TYPE ST_CX_EtherCATMasterState :
STRUCT
	arrADSAddr		: ARRAY[0..5] OF BYTE;
	nState			: UINT;
	nDevID			: UINT;
	nSlaveCount		: UINT;
	nDevState		: UINT;
END_STRUCT
END_TYPE

(* stored: Version 1.1.0.1
   DUT ST_CX_EtherCATMasterState: Id {6a9a4ff2-44c3-47cf-b322-4ac167820a99} *)
